PROGRAM POU
VAR
END_VAR

END_PROGRAM

(* stored: Version 1.1.0.1, ProductVersion 3.1.4023.21
   POU POU: Id {8ae29ff4-6456-4425-8b4c-cc2f9da92797}, SpecialFunc None *)
